{attribute 'GeneratedUsingTerminal: EL2212-0000-0018'}
{attribute addProperty BoxType "EL2212-0000-0018"}
{attribute addProperty Id "Ready_to_activateBOOL1Output_activeBOOL1Tristate_activeBOOL1WarningBOOL1ErrorBOOL1Sync_errorBOOL1TxPDO_ToggleBOOL1"}
{attribute addProperty CRC "3655113755"}
{attribute addProperty Size "7"}
TYPE Status_D9DC9C1B :
STRUCT
	{attribute addProperty Name "Ready_to_activate"}
	Ready_to_activate : BOOL;
	{attribute addProperty Name "Output_active"}
	Output_active : BOOL;
	{attribute addProperty Name "Tristate_active"}
	Tristate_active : BOOL;
	{attribute addProperty Name "Warning"}
	Warning : BOOL;
	{attribute addProperty Name "Error"}
	Error : BOOL;
	{attribute addProperty Name "Sync_error"}
	Sync_error : BOOL;
	{attribute addProperty Name "TxPDO_Toggle"}
	TxPDO_Toggle : BOOL;
END_STRUCT
END_TYPE

(* stored: Version 1.2.0.0, ProductVersion 3.1.4024.9
   DUT Status_D9DC9C1B: Id {79072d0a-7028-4072-92b0-eb5cf9f932b2} *)
